{attribute addProperty BoxType "EJ6002-0000-0016"}
{attribute addProperty Id "COM_Inputs_ChannelAT %I*ARRAY[0..23] OF COM_Inputs_Channel_85D1D733384480COM_Outputs_ChannelAT %Q*ARRAY[0..23] OF COM_Outputs_Channel_85BCA431384480WcStateAT %I*WcState_98A4DF7520.250InfoDataAT %I*InfoData_BC63D37F80100"}
{attribute addProperty CRC "226543692"}
{attribute addProperty SizeInBites "850"}
{attribute addProperty SizeInBytes "106.25"}
TYPE EJ6002_880A624E :
STRUCT
	{attribute addProperty Name "COM_Inputs_Channel"}
	COM_Inputs_Channel : ARRAY[0..23] OF COM_Inputs_Channel_85D1D733;
	{attribute addProperty Name "COM_Outputs_Channel"}
	COM_Outputs_Channel : ARRAY[0..23] OF COM_Outputs_Channel_85BCA431;
	{attribute addProperty Name "WcState"}
	WcState : WcState_98A4DF75;
	{attribute addProperty Name "InfoData"}
	InfoData : InfoData_BC63D37F;
END_STRUCT
END_TYPE

(* stored: Version 1.2.0.0, ProductVersion 3.1.4024.9
   DUT EJ6002_880A624E: Id {a283454f-88c2-4426-b89b-c5cfa1e99fe1} *)
